% RSLogix 500 project reject_tracking_parky_timer.RSS, saved by version 8.30.00.16 %
PROJECT "UNTITLED"    % processor: Bul.1763 MicroLogix 1100 Series B %

PROGRAM FILES
  LAD 2   10 rungs

DATA FILES
  O0 OUTPUT  4 elements
  I1 INPUT  6 elements
  S2 STATUS  66 elements
  B3 BINARY  1 elements
  T4 TIMER  2 elements
  C5 COUNTER  1 elements
  R6 CONTROL  1 elements
  N7 INTEGER  1 elements
  F8 FLOAT  1 elements
  B9 INPUT_BFFR  1 elements
  N10 CONSTANCE  10 elements
  B11 RJECT_FIFO  256 elements

LADDER 2
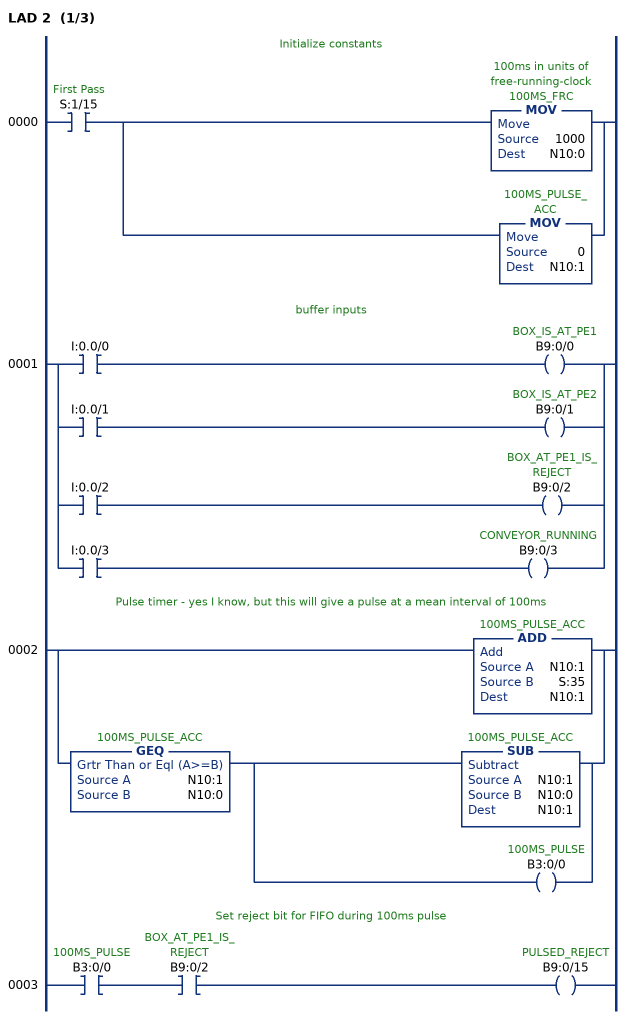
% Rung: 0 %
% Initialize constants %
SOR XIC S:1/15 BST MOV 1000 N10:0 NXB MOV 0 N10:1 BND EOR
%   S:1/15  "First Pass" %
%   N10:0  100MS_FRC  "100ms in units of free-running-clock" %
%   N10:1  100MS_PULSE_ACC %
% Rung: 1 %
% buffer inputs %
SOR BST XIC I:0.0/0 OTE B9:0/0 NXB XIC I:0.0/1 OTE B9:0/1 NXB XIC I:0.0/2 OTE B9:0/2 NXB XIC I:0.0/3 OTE B9:0/3 BND EOR
%   B9:0/0  BOX_IS_AT_PE1 %
%   B9:0/1  BOX_IS_AT_PE2 %
%   B9:0/2  BOX_AT_PE1_IS_REJECT %
%   B9:0/3  CONVEYOR_RUNNING %
% Rung: 2 %
% Pulse timer - yes I know, but this will give a pulse at a mean interval of 100ms %
SOR BST ADD N10:1 S:35 N10:1 NXB GEQ N10:1 N10:0 BST SUB N10:1 N10:0 N10:1 NXB OTE B3:0/0 BND BND EOR
%   N10:1  100MS_PULSE_ACC %
%   S:35  "Last 1 ms Scan Time" %
%   N10:0  100MS_FRC  "100ms in units of free-running-clock" %
%   B3:0/0  100MS_PULSE %
% Rung: 3 %
% Set reject bit for FIFO during 100ms pulse %
SOR XIC B3:0/0 XIC B9:0/2 OTE B9:0/15 EOR
%   B3:0/0  100MS_PULSE %
%   B9:0/2  BOX_AT_PE1_IS_REJECT %
%   B9:0/15  PULSED_REJECT %

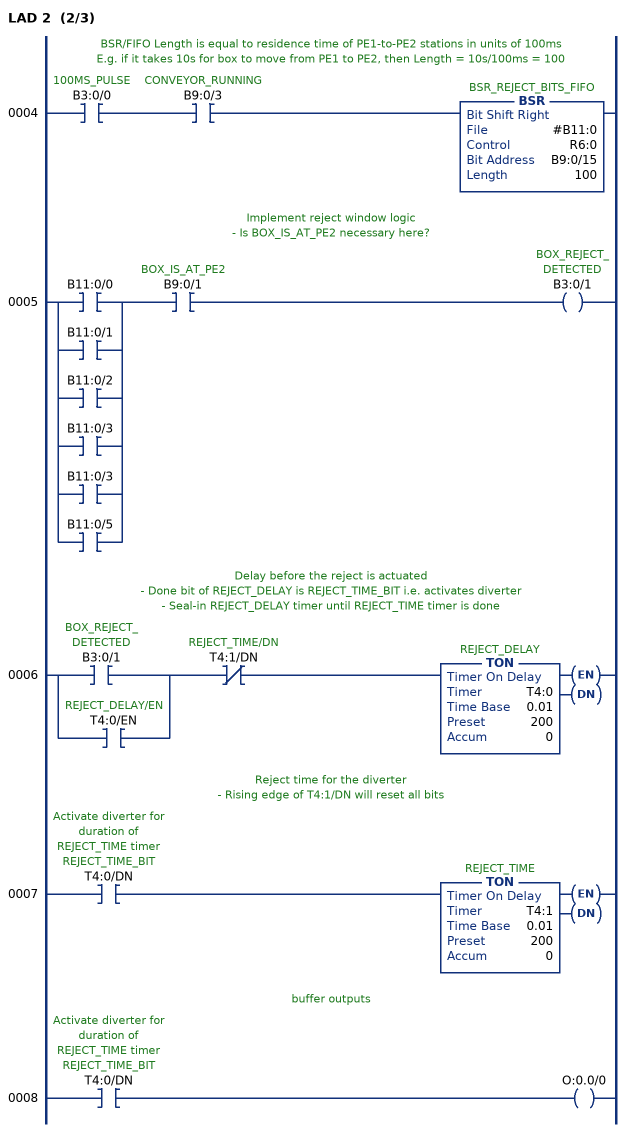
% Rung: 4 %
% BSR/FIFO Length is equal to residence time of PE1-to-PE2 stations in units of 100ms
% E.g. if it takes 10s for box to move from PE1 to PE2, then Length = 10s/100ms = 100 %
SOR XIC B3:0/0 XIC B9:0/3 BSR #B11:0 R6:0 B9:0/15 100 EOR
%   B3:0/0  100MS_PULSE %
%   B9:0/3  CONVEYOR_RUNNING %
%   B11:0  BSR_REJECT_BITS_FIFO %
%   R6:0  BSR_REJECT_FIFO %
%   B9:0/15  PULSED_REJECT %
% Rung: 5 %
% Implement reject window logic
% - Is BOX_IS_AT_PE2 necessary here? %
SOR BST XIC B11:0/0 NXB XIC B11:0/1 NXB XIC B11:0/2 NXB XIC B11:0/3 NXB XIC B11:0/3 NXB XIC B11:0/5 BND XIC B9:0/1 OTE B3:0/1 EOR
%   B9:0/1  BOX_IS_AT_PE2 %
%   B3:0/1  BOX_REJECT_DETECTED %
% Rung: 6 %
% Delay before the reject is actuated
% - Done bit of REJECT_DELAY is REJECT_TIME_BIT i.e. activates diverter
% - Seal-in REJECT_DELAY timer until REJECT_TIME timer is done %
SOR BST XIC B3:0/1 NXB XIC T4:0/EN BND XIO T4:1/DN TON T4:0 0.01 200 0 EOR
%   B3:0/1  BOX_REJECT_DETECTED %
%   T4:0  REJECT_DELAY %
%   T4:1  REJECT_TIME %
% Rung: 7 %
% Reject time for the diverter
% - Rising edge of T4:1/DN will reset all bits %
SOR XIC T4:0/DN TON T4:1 0.01 200 0 EOR
%   T4:0/DN  REJECT_TIME_BIT  "Activate diverter for duration of REJECT_TIME timer" %
%   T4:1  REJECT_TIME %
% Rung: 8 %
% buffer outputs %
SOR XIC T4:0/DN OTE O:0.0/0 EOR
%   T4:0/DN  REJECT_TIME_BIT  "Activate diverter for duration of REJECT_TIME timer" %

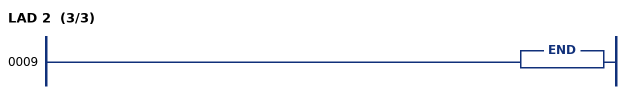
% Rung: 9 %
SOR END EOR

DATA TABLE (non-zero values as saved)
DATA T4
% .PRE .ACC %
% T4:0 % 200 0
% T4:1 % 200 0
DATA R6
% .LEN .POS %
% R6:0 % 100 0
